// TIA Portal V20 export
TYPE "LER_typeHotWireCutterMonitoring"
// stored: Access Published
   STRUCT
      on : Bool;
      off : Bool;
   END_STRUCT;
END_TYPE
